FUNCTION_BLOCK Resetting_State  IMPLEMENTS ITF_State
VAR_INPUT
END_VAR
VAR_OUTPUT
END_VAR
VAR
	pPML_Base : POINTER TO PML_StatePattern_Base;
	_stateMachine : IPmlStateMachine;
END_VAR

METHOD Cycle : BOOL
VAR_INPUT
END_VAR
_stateMachine.SetStateComplete();
pPML_Base^.SetState(pPML_Base^.idle);
END_METHOD

METHOD FB_init : BOOL
VAR_INPUT
	bInitRetains : BOOL; // if TRUE, the retain variables are initialized (warm start / cold start)
	bInCopyCode : BOOL;  // if TRUE, the instance afterwards gets moved into the copy code (online change)
	pPML_Base : POINTER TO PML_StatePattern_Base;
	statemachine : IPmlStateMachine;
END_VAR
_stateMachine := statemachine;
THIS^.pPML_Base := pPML_Base;
END_METHOD

END_FUNCTION_BLOCK

(* stored: Version 1.1.0.1, ProductVersion 3.1.4024.12
   POU Resetting_State: Id {04a20e74-9cab-4680-bae9-bdaebe1065f6}, SpecialFunc None
   Method Cycle: Id {052db35b-c879-47af-ae1f-f617fd56c725}
   Method FB_init: Id {5542bb07-3bcc-4a67-9f96-d403aa82b034} *)
